TYPE ST_ProcessDiag :
STRUCT
    bSPD01Fault              	  : BOOL;

    bPauseRequiredByProcess       : BOOL;
    bPauseNoLime                  : BOOL;
    bPauseNoPerlite               : BOOL;

    bSystemReady				  : BOOL;
END_STRUCT
END_TYPE

(* stored: Version 1.1.0.1, ProductVersion 3.1.4024.16
   DUT ST_ProcessDiag: Id {84b875d8-993a-4fd8-944d-641be00b212d} *)
